(* CoDeSys 2.3 export: FUN_KD2.EXP *)

(* POU PRG/Fun_KD2, ST *)
PROGRAM Fun_KD2
VAR
	Fun : DRIVE;
	CMD_FanRunLatch : BOOL := FALSE;


END_VAR
	(* Если активирован ручной режим управления вентилятором КД2 *)
	IF NOT KD2.FAN.xMode_AUTO THEN
		KD2.FAN.xCMD_RUN := (KD2.FAN.xBtnRun OR CMD_FanRunLatch )
									AND NOT (KD2.FAN.xBtnStop);
	END_IF;

	CMD_FanRunLatch := KD2.FAN.xCMD_RUN;
END_PROGRAM
